Staubli VAL3: loadmaster5.pgx

program loadmaster5(string x_sMasterFile5 (dimensions=1))
begin
  if master:libLoad(x_sMasterFile5)<0
    popUpMsg("nO ok")
  endIf
  frmaster[5].trsf=master:tTool.trsf
  //取个数
  nsize[5]=size(master:ptRoutingPath)
  //存个数
  resize(pdemo5,1,nsize[5])
  //保存程序
  master:libSave()
end
